PROGRAM MAIN
VAR
	fbFileLoggerFactory	  : FB_FileLoggerFactory('File.csv');
	refFileLoggerFactory  : REFERENCE TO FB_FileLoggerFactory := fbFileLoggerFactory;
	fbLogger 			  : FB_Logger(refFileLoggerFactory);	
	sRetMsg				  : STRING;
END_VAR

sRetMsg := fbLogger.Write('Hello');

END_PROGRAM

(* stored: Version 1.1.0.1, ProductVersion 3.1.0.24
   POU MAIN: Id {fd6e49ae-9c60-4ba4-ba01-45f20a4b6c2c} *)
